FUNCTION_BLOCK PistonOutputLogic
VAR
	timer: TOF;
	timerElapsed: BOOL;
	riseTrig: R_TRIG;
	riseTrigDetected: BOOL;
END_VAR

timer(IN := gvl.SwitchTableExit, PT := T#0.5S, Q => timerElapsed);
//riseTrig(CLK := gvl.SwitchTableExit, Q => riseTrigDetected);

IF timerElapsed THEN
	gvl.PistonOutputBackwards := FALSE;
	gvl.PistonOutputForward := TRUE;
	gvl.MotorBeltMove := TRUE;
ELSE
	gvl.PistonOutputBackwards := TRUE;
	gvl.PistonOutputForward := FALSE;
END_IF

//IF riseTrigDetected THEN
//	LocalVariables.Locations[5].Item.Id := LocalVariables.Locations[4].Item.Id;
//	LocalVariables.Locations[5].Item.Recipe := LocalVariables.Locations[4].Item.Recipe;
//	LocalVariables.Locations[4].Item.Id := NULL;
//	LocalVariables.Locations[4].Item.Recipe := LocalVariables.Recipe;
//END_IF

END_FUNCTION_BLOCK

(* stored: Version 1.1.0.1, ProductVersion 3.1.4024.12
   POU PistonOutputLogic: Id {3ca4cc8a-59a8-49d1-bcf1-188defb0c6a9}, SpecialFunc None *)
